PROGRAM PR_Line01
VAR PERSISTENT
//----------------VAR SETTING--------------------
	timerCheckCylinder_Up			: REAL;//CupSupply
	timerCheckCylinder_Dw			: REAL;
	timerCheckEmpty					: REAL;
	timerCheckStuck					: REAL;
	timerCylinder_Up_extend 		: REAL;
	timerCylinder_Suction_Cup_extend: REAL;
	timerCylinder_Suction_Cup		: REAL;
	timerCylinder_Suction_Val		: REAL;
	timerCylinder_Suction_pick		: REAL;
	fSpeed_motor_mixer				: REAL;//FoodMixer
	fTimer_Reverse					: REAL;
	fFast_Speed						: REAL;//FoodWeight
	fSlow_Speed_1					: REAL;
	fSlow_Speed_2					: REAL;
	fDerisedWeight_Food				: REAL;
	fChangeMode_Food_1				: REAL;
	fChangeMode_Food_2				: REAL;
	fMaxWeight_Food					: REAL;
	fPerStop_Food					: REAL;
	fTimer_Food						: REAL;
	fTimer_Alarm_Food				: REAL;
	fTimer_Check_Food				: REAL;
	fDelta_Food						: REAL;
	fTimer_rever_food				: REAL;
	fTimer_Error_Food				: REAL;
	fFast_Speed_vibrating_funnel	: REAL;//WormWeight
	fSlow_Speed_vibrating_funnel_1	: REAL;
	fSlow_Speed_vibrating_funnel_2	: REAL;
	fDerisedWeight_Worm				: REAL;
	fChangeMode_Worm_1				: REAL;
	fChangeMode_Worm_2				: REAL;
	fMaxWeight_Worm					: REAL;
	fPerStop_Worm					: REAL;
	fTimer_Worm						: REAL;
	fTimer_Alarm_Worm				: REAL;
	fTimer_Check_Worm				: REAL;
	fTimer_Check_Cylinder			: REAL;
	fDelta_Worm						: REAL;
	fTimer_Error_Worm				: REAL;
	timerCylinder_Suction			: REAL;//LidSupply
	timerCheckLidRelease			: REAL;
	timerLidBlow					: REAL;
	timerCheckLidEmpty				: REAL;
	timerCheckLidSuck				: REAL;
	timerCylinder_Stopper			: REAL;
	timer_Check_Cylinder_extend		: REAL;//LidClose
	timer_Check_Cylinder_retract	: REAL;
	timer_CloseLid					: REAL;
	fTimer_Comb						: REAL;//Transfer
	fTimer_Clip						: REAL;
	fTimer_Move_Comb				: REAL;
//-----------------VAR HMI-------------------
	fProductLog						: ARRAY [1..2] OF ARRAY  [1..5] OF REAL;
END_VAR

VAR
	bStatus_Food					: BOOL;
	bStatus_Worm					: BOOL;
//----------------VAR MANUAL---------------------
	bCylinder_up_extend 			: BOOL;//CupSupply
	bCylinder_up_retract 			: BOOL;
	bCylinder_dw_extend 			: BOOL;
	bCylinder_dw_retract 			: BOOL;
	bCylinder_Suction_cup_extend	: BOOL;
	bCylinder_Suction_cup_retract	: BOOL;
	bUp_Motor_Mixer					: BOOL;//FoodMixer
	bDown_Motor_Mixer				: BOOL;
	bMotor_mixer_Manual				: BOOL;
	bMotor_mixer_reverse			: BOOL;
	bUp_Food_Motor					: BOOL;//FoodWeight
	bDown_Food_Motor				: BOOL;
	bZero_Loadcell_Food				: BOOL;
	bMotor_Food						: BOOL;
	bMotor_Food_reverse				: BOOL;
	bUp_vibrating_funnel			: BOOL;//WormWeight
	bDown_vibrating_funnel			: BOOL;
	bZero_Loadcell_Worm				: BOOL;
	bCylinder_Block_Worm_Extend		: BOOL;
	bCylinder_Block_Worm_Retract	: BOOL;
	bMotor_vibrating_funnel			: BOOL;	
	bCylinder_LidStopper_extend 	: BOOL;//LidSupply
	bCylinder_LidStopper_retract 	: BOOL;
	bCylinder_Suction_extend		: BOOL;
	bCylinder_Suction_retract		: BOOL;
	bLidSuctionValve				: BOOL;
	bCupSuctionValve				: BOOL;
	bBlowValve						: BOOL;
	bCylinder_CloseLid_Extend		: BOOL;//LidClose
	bCylinder_CloseLid_Retract		: BOOL;
	bCylinder_Comb_Extend			: BOOL;//Transfer
	bCylinder_Comb_Retract			: BOOL;
	bCylinder_Clip_Extend			: BOOL;
	bCylinder_Clip_Retract			: BOOL;
	bCylinder_Move_Comb_Extend		: BOOL;
	bCylinder_Move_Comb_Retract		: BOOL;
//------------------fbmodule----------------
	fb_CupSupply	: FB_CupSupplyModule;
	fb_FoodMixer	: FB_FoodMixerModule;
	fb_FoodWeight	: FB_FoodWeightModule;
	fb_WormWeight	: FB_WormWeightModule;
	fb_LidSupply	: FB_LidSupplyModule;
	fb_LidClose		: FB_LidCloseModule;
	fb_Transfer		: FB_Transfer;
//---------------- VAR Method ---------------
	nState				: INT;
	nState_Dropcup		: INT;
	nState_Transfer		: INT;
	nState_FoodWeight	: INT;
	nState_WormWeight	: INT;
	nState_LidClose		: INT;
	nState_LidSupply	: INT;
	nDoneTransfer		: INT;
	nDoneTransferStop	: INT;
	tmp					: INT;
	bDoneTakeLid		: BOOL;
	bDoneTransfer		: BOOL;
	bDoneCupSupply		: BOOL;
	bDoneFoodWeight		: BOOL;
	bDoneWormWeight		: BOOL;
	bDoneLidSupply		: BOOL;
	bDoneLidClose		: BOOL;
	bEnable				: BOOL;
	bFinishCupSupply	: BOOL;
	bFinishFoodWeight	: BOOL;
	bFinishWormWeight	: BOOL;
	bFinishLidSupply	: BOOL;
	bFinishLidClose		: BOOL;
	bFinishTransfer		: BOOL;
	//-------VAR--------------
	nStateConveyor		: INT;
	fbtimertransfer		: TON;
	nStateStop			: INT;
	fbTimer				: ton;
	fbtimerStop			: ton;
	fbTimerCycle		: ton;
	timeCycle			: REAL :=1;
	fproduct			: INT;
	nstateCycle			: INT;
	bDone				: R_TRIG;
	fbDelay				: TON;
	bStatus_Food_order	: ARRAY [1..3] OF BOOL;
	bStatus_Worm_order	: ARRAY [1..3] OF BOOL;
	bStatus_Lid_order	: ARRAY [1..3] OF BOOL;
	i1,i2,i3			: INT := 0;
	xathucan			: BOOL;
	xasau				: BOOL;
	daothucan			: BOOL;
	transfer			: BOOL;
	nstatetest1			: INT;
	nstatetest2			: INT;
	nstatetest3			: INT;
	nstatetest4         : INT;
	bxa					: BOOL;
	bCheck				: BOOL;
	bypassfood			: BOOL;
	bypassWorm			: BOOL;
	bypassLid			: BOOL;
	eles: INT;
END_VAR

fb_CupSupply(
	nLine:= 1 , 
	timerCheckCylinder_Up:= timerCheckCylinder_Up, 
	timerCheckCylinder_Dw:= timerCheckCylinder_Dw, 
	timerCheckEmpty:= timerCheckEmpty, 
	timerCheckStuck:= timerCheckStuck,
	timerCylinder_Up_extend := timerCylinder_Up_extend,
	timerCylinder_Suction:= timerCylinder_Suction_Cup,
	timerCylinder_Suction_extend:= timerCylinder_Suction_Cup_extend,
	ttimerCylinder_val:= timerCylinder_Suction_Val,
	timerCylinder_Suction_pick:= timerCylinder_Suction_pick);

fb_FoodMixer(
	nLine:= 1,
	UnitID:= 4, 
	fSpeed_motor_mixer:= fSpeed_motor_mixer,
	fTimer_Reverse:= fTimer_Reverse);
		
fb_FoodWeight(
	nLine:= 1, 
	UnitID:= 7, 
	fFast_Speed:= fFast_Speed, 
	fSlow_Speed_1:= fSlow_Speed_1, 
	fSlow_Speed_2:= fSlow_Speed_2, 
	fDerisedWeight_Food:= fDerisedWeight_Food, 
	fChangeMode_Food_1:= fChangeMode_Food_1, 
	fChangeMode_Food_2:= fChangeMode_Food_2, 
	fMaxWeight_Food:= fMaxWeight_Food, 
	fPerStop_Food:= fPerStop_Food, 
	fTimer_Food:= fTimer_Food, 
	fTimer_Alarm_Food:= fTimer_Alarm_Food, 
	fTimer_Check_Food:= fTimer_Check_Food, 
	fDelta_Food:= fDelta_Food,
	fTimer_Reverse := fTimer_rever_food,
	fTimer_Error_Food := fTimer_Error_Food, 
	fProductLogF=> fProductLog[1],
	bStatus_Food=> bStatus_Food,
	Time_start => Time_Start_Food_line1,
	Time_Stop => Time_Stop_Food_line1,
	status=>bStatus_Food_line1,
	fweight_iot =>fWeight_food_line1);

fb_LidClose(
	nLine:= 1, 
	timer_Check_Cylinder_extend:= timer_Check_Cylinder_extend, 
	timer_Check_Cylinder_retract:= timer_Check_Cylinder_retract, 
	timer_CloseLid:= timer_CloseLid);
	
fb_LidSupply(
	nLine:= 1, 
	timerCylinder_Suction:= timerCylinder_Suction, 
	timerCheckLidRelease:= timerCheckLidRelease, 
	timerLidBlow:= timerLidBlow, 
	timerCheckLidEmpty:= timerCheckLidEmpty, 
	timerCheckLidSuck:= timerCheckLidSuck, 
	timerCylinder_Stopper:= timerCylinder_Stopper);

fb_Transfer(
	nLine:= 1, 
	fTimer_Comb:= fTimer_Comb, 
	fTimer_Clip:= fTimer_Clip, 
	fTimer_Move_Comb:= fTimer_Move_Comb, 
	nDoneTransfer=> nDoneTransfer,
	bDoneTransfer=> bDoneTransfer);

fb_WormWeight(
	nLine:= 1, 
	UnitID:= 5, 
	fFast_Speed_vibrating_funnel:= fFast_Speed_vibrating_funnel, 
	fSlow_Speed_vibrating_funnel_1:= fSlow_Speed_vibrating_funnel_1, 
	fSlow_Speed_vibrating_funnel_2:= fSlow_Speed_vibrating_funnel_2, 
	fDerisedWeight_Worm:= fDerisedWeight_Worm, 
	fChangeMode_Worm_1:= fChangeMode_Worm_1, 
	fChangeMode_Worm_2:= fChangeMode_Worm_2, 
	fMaxWeight_Worm:= fMaxWeight_Worm, 
	fPerStop_Worm:= fPerStop_Worm, 
	fTimer_Worm:= fTimer_Worm, 
	fTimer_Alarm_Worm:= fTimer_Alarm_Worm, 
	fTimer_Check_Worm:= fTimer_Check_Worm, 
	fTimer_Check_Cylinder:= fTimer_Check_Cylinder, 
	fDelta_Worm:= fDelta_Worm,
	fTimer_Error_Worm:= fTimer_Error_Worm, 
	fProductLog=> fProductLog[2],
	bStatus_Worm=>bStatus_Worm,
	Time_start=>Time_Start_Worm_line1,
	Time_Stop=>Time_Stop_Worm_line1,
	status=>bStatus_Worm_line1,
	fweight_iot =>fWeight_Worm_line1);

IF bClear1 THEN
	nResult_false1 := 0;
	nResult_true1 := 0;
	nCount1 := 0;
	bClear1 := FALSE;
END_IF	

fDerisedWeight_Food_line1	:= fDerisedWeight_Food;
fDerisedWeight_Worm_line1	:= fDerisedWeight_Worm;
fActDelta_Food_line1		:= fb_FoodWeight.fActDelta_Food;
fActDelta_Worm_line1		:= fb_WormWeight.fActDelta_Worm;
fDelta_Food_line1			:= fb_FoodWeight.fDelta_Food;
fDelta_Worm_line1			:= fb_WormWeight.fDelta_Worm;
	
IF getuser = 'Operator' THEN
	bypassfood := FALSE;
	bypassWorm := FALSE;
END_IF

ACTION Auto:
CASE nState OF
	0:// int
		bStatus_Food_order[1] := FALSE;
		bStatus_Worm_order[1] := FALSE;
		bStatus_Lid_order[1]  := FALSE;
		fb_Transfer.Init();
		fb_FoodWeight.SetZero();
		fb_WormWeight.SetZero();
		nDoneTransferStop	  := 0;
		i1 		:= 0;
		i2 		:= 0;
		i3 		:= 0;
		bfinish1	:= TRUE;
		nState 	:= 1;
		
	1: // Start
		nState_FoodWeight := 0;
		nState_WormWeight := 0;
		nState_LidSupply := 0;
		nState_LidClose := 0;
		bResetAuto1			:= FALSE;
		bDoneCupSupply 		:= FALSE;
		bDoneFoodWeight 	:= FALSE;
		bDoneWormWeight 	:= FALSE;
		bDoneLidSupply 		:= FALSE;
		bDoneLidClose 		:= FALSE;
		fb_FoodWeight.SetZero();
		fb_WormWeight.SetZero();
		nState := 11;
	11:
		bResetAuto1			:= FALSE;
		nState_Dropcup := 0;
		nState_Transfer := 0;
		bStop1 := FALSE;
		bShift_is_over1 := FALSE;
		bStatusStart1 := FALSE;
		fb_FoodMixer.Stop();
		nStatus1	:= 'STOP';
		bFinishCupSupply 	:= FALSE;
		bFinishFoodWeight 	:= FALSE;
		bFinishWormWeight	:= FALSE;
		bFinishLidSupply	:= FALSE;
		bFinishLidClose		:= FALSE;
		bFinishTransfer		:= FALSE;
		bfinish1	:= TRUE;
		nState := 22;
	22:
		IF bStart1 THEN
			bfinish1		:= FALSE;
			bStatusStart1 	:= TRUE;
			bToDropcup1 	:= FALSE;
			bResetAuto1		:= TRUE;
			status			:= 'RUN';
			nState := 2;
		END_IF
		
	2: // start mode auto
		bfinish1		:= FALSE;
		nStatus1	:= 'RUN';
		bResetAuto1		:= TRUE;
		bStart1 := FALSE;
		IF bypassfood THEN
			fb_FoodMixer.Stop();
		ELSE
			fb_FoodMixer.Auto();
		END_IF
		fb_CupSupply.CheckCup();
		fb_LidSupply.CheckLid();
		bDone(CLK := bDoneTransfer);
		CASE nstateCycle OF 
			0:
				fbTimerCycle(IN := TRUE, PT := T#100S);
				IF bDone.Q THEN
					nstateCycle := 1;
				END_IF
			1:
				timeCycle := TIME_TO_REAL(fbTimerCycle.ET)/1000;
				nstateCycle := 2;
			2: 
				fproduct :=  REAL_TO_INT(3600/(timeCycle+0.001));
				fbTimerCycle(IN := FALSE);
				nstateCycle := 0;
		END_CASE
		CASE nState_Dropcup OF
			0:// waiting for transfer
				fbDelay(IN := FALSE);
				fb_CupSupply.HoldCup();
				IF bToDropcup1 THEN
					nState_Dropcup := 1;
				END_IF
			1:// dropcup
				IF fb_CupSupply.DropCup() THEN
					bDoneCupSupply := TRUE;
					bToDropcup1 := FALSE;
					nState_Dropcup := 2;
				END_IF
			2:
				fbDelay(IN := TRUE, PT := T#300MS);
				IF fbDelay.Q THEN
					nState_Dropcup := 0;
				END_IF
		END_CASE
		
		CASE nState_FoodWeight OF
			0:// waiting for transfer
				IF bDoneTransfer THEN
					i1 := i1 + 1;
					fbTimer(IN := FALSE);
					nState_FoodWeight := 1;	
				END_IF
			1:// Check cup present
				IF NOT fb_FoodWeight.bIsCupPresent THEN
					IF bypassfood THEN
						nState_FoodWeight := 3;
						bStatus_Food_order[i1] := TRUE;
					ELSE
						nState_FoodWeight := 2;
					END_IF
				ELSE
					bStatus_Food_order[i1] := FALSE;
					nState_FoodWeight := 3;
				END_IF
			2:// FoodWeight
				IF NOT fb_FoodWeight.bIsCupPresent THEN
					IF fb_FoodWeight.Auto() THEN
						bStatus_Food_order[i1] := bStatus_Food;
						nState_FoodWeight := 3;
					END_IF
				ELSE
					nState_FoodWeight := 22;
				END_IF 
			22:
				fbTimer(IN := TRUE, PT := T#0.3S);
				fb_FoodWeight.Auto();
				IF fbTimer.Q THEN
					fb_FoodWeight.Init();
					nState_FoodWeight := 0;
				END_IF
			3:// check i
				IF i1 < 3 THEN
					nState_FoodWeight := 5;
				ELSE 
					i1 := 2;
					nState_FoodWeight := 4;
				END_IF
			4:// dao vi tri
				bStatus_Food_order[1] := bStatus_Food_order[2];
				bStatus_Food_order[2] := bStatus_Food_order[3];
				nState_FoodWeight := 5;
			5:// Done
				bDoneFoodWeight := TRUE;
				nState_FoodWeight := 10;
		END_CASE
		
		CASE nState_WormWeight OF
			0: // waiting for transfer
				IF bDoneTransfer THEN
					i2 := i2 + 1;;
					fbTimer(IN := FALSE);
					nState_WormWeight := 1;
				END_IF
			1:
				IF NOT fb_WormWeight.bIsCupPresent THEN
					nCount1 := nCount1 + 1;
					nState_WormWeight := 11;
				ELSE
					bStatus_Worm_order[i2] := FALSE;
					nState_WormWeight := 3;
				END_IF
			11: // check food
				IF bStatus_Food_order[1] THEN
					IF bypassWorm THEN
						nState_WormWeight := 3;
						bStatus_Worm_order[i2] := TRUE;
					ELSE
						nState_WormWeight := 2;
					END_IF
				ELSE
					bStatus_Worm_order[i2] := FALSE;
					nState_WormWeight := 3;
				END_IF	
			2:// WormWeight
				IF NOT fb_WormWeight.bIsCupPresent THEN
					IF fb_WormWeight.Auto() THEN
						bStatus_Worm_order[i2] := bStatus_Worm;
						nState_WormWeight := 3;
					END_IF
				ELSE
					nState_WormWeight := 22;
				END_IF
			22:
				fbTimer(IN := TRUE, PT := T#0.3S);
				fb_WormWeight.Auto(); 
				IF fbTimer.Q THEN
					fb_WormWeight.Init();
					nState_WormWeight := 0;
				END_IF
			3:// check i
				IF bStatus_Worm_order[i2] THEN
					nResult_true1 := nResult_true1 + 1;
				END_IF
				IF i2 < 3 THEN
					nState_WormWeight := 5;
				ELSE
					i2 := 2;
					nState_WormWeight := 4;
				END_IF
			4:// dao vi tri
				nResult_false1 := nCount1 - nResult_true1;
				bStatus_Worm_order[1] := bStatus_Worm_order[2];
				bStatus_Worm_order[2] := bStatus_Worm_order[3];
				nState_WormWeight 	  := 5;
			5:// Done 
				bDoneWormWeight       := TRUE;
				nState_WormWeight	  := 10;
		END_CASE
		
		CASE nState_LidSupply OF
			0:// waiting for transfer
				IF bDoneTransfer THEN
					i3 := i3 + 1;
					nState_LidSupply := 1;
				END_IF
			1:// check worm
				IF bStatus_Worm_order[1] THEN
					IF bypassLid THEN
						bStatus_Lid_order[i3] := FALSE;
						nState_LidSupply := 4;
					ELSE
						nState_LidSupply := 2;
					END_IF
				ELSE
					bStatus_Lid_order[i3] := FALSE;
					nState_LidSupply := 4;
				END_IF
			2:// take lid
				IF fb_LidSupply.TakeLid() THEN
					nState_LidSupply := 3;
				END_IF
			3:// drop lid
				IF fb_LidSupply.DropLid() THEN
					bStatus_Lid_order[i3] := TRUE;
					nState_LidSupply := 4;
				END_IF
			4:// check i
				IF i3 < 3 THEN
					nState_LidSupply := 6;
				ELSE
					i3 := 2;
					nState_LidSupply := 5;
				END_IF
			5:// dao vi tri
				bStatus_Lid_order[1] := bStatus_Lid_order[2];
				bStatus_Lid_order[2] := bStatus_Lid_order[3];
				nState_LidSupply 	 := 6;
			6:// Done
				bDoneLidSupply 		 := TRUE;
				nState_LidSupply 	 := 10;
		END_CASE
		
		CASE nState_LidClose OF
			0: // waiting for transfer
				IF bDoneTransfer THEN
					nState_LidClose := 1;
				END_IF
			1:// Check lid supply
				IF  bStatus_Lid_order[1] THEN
					nState_LidClose := 2;
				ELSE
					nState_LidClose := 3;
				END_IF
			2:// Close lid
				IF fb_LidClose.CloseLid() THEN
					nState_LidClose := 3;
				END_IF
			3://Done
				bDoneLidClose := TRUE;
				nState_LidClose := 10;
		END_CASE
		
		CASE nState_Transfer OF
			0:// waiting for Done module
				IF nDoneTransfer = 0 THEN
					nState_Transfer := 1;
				ELSIF nDoneTransfer > 0 THEN
					IF bDoneCupSupply AND bDoneFoodWeight AND bDoneWormWeight AND bDoneLidSupply AND bDoneLidClose THEN
						nState_Transfer := 1;
					END_IF
				END_IF
			1:
				IF fb_CupSupply.isCupDrop THEN
					bDoneCupSupply 	:= FALSE;
					bDoneFoodWeight := FALSE;
					bDoneWormWeight := FALSE;
					bDoneLidSupply 	:= FALSE;
					bDoneLidClose 	:= FALSE;
					nState_Transfer := 11;
				ELSE 
					F_SetError(2,nLine:=1);
				END_IF
			11:// transfer
				IF fb_Transfer.Auto() THEN
					nShoot1 := nShoot1 + 1; 
					nState_Transfer:= 2;
				END_IF
			2:
				nState_FoodWeight := 0;
				nState_WormWeight := 0;
				nState_LidSupply  := 0;
				nState_LidClose	  := 0;
				nState_Transfer	  := 0;
		END_CASE
		//Stop button
		IF bStop1 THEN
			nState := 3;
			bStartLine1 := FALSE;
		ELSIF bShift_is_over1 THEN
			nState := 4;
		END_IF
	3://Stop
		bfinish1 := FALSE;
		fb_CupSupply.CheckCup();
		fb_LidSupply.CheckLid();
		bResetAuto1		:= TRUE;
		nStatus1	:= 'RUN';
		IF bypassfood THEN
			fb_FoodMixer.Stop();
		ELSE
			fb_FoodMixer.Auto();
		END_IF
		CASE nState_Dropcup OF
			0:// waiting for transfer
				fbDelay(IN := FALSE);
				fb_CupSupply.HoldCup();
				IF bToDropcup1 THEN
					nState_Dropcup := 1;
				END_IF
				IF bFinishTransfer THEN
					nState_Dropcup := 10;
				END_IF
			1:// dropcup
				IF fb_CupSupply.DropCup() THEN
					bDoneCupSupply := TRUE;
					bToDropcup1 := FALSE;
					nState_Dropcup := 2;
				END_IF
			2:
				fbDelay(IN := TRUE, PT := T#300MS);
				IF fbDelay.Q THEN
					nState_Dropcup := 10;
				END_IF
			10:// finish
				bDoneCupSupply := TRUE;
				bFinishCupSupply := TRUE;
		END_CASE
		
		CASE nState_FoodWeight OF
			0:// waiting for transfer
				IF bDoneTransfer THEN
					i1 := i1 + 1;
					fbTimer(IN := FALSE);
					nState_FoodWeight := 1;	
				END_IF
			1:// Check cup present
				IF NOT fb_FoodWeight.bIsCupPresent THEN
					IF bypassfood THEN
						nState_FoodWeight := 3;
						bStatus_Food_order[i1] := TRUE;
					ELSE
						nState_FoodWeight := 2;
					END_IF
				ELSE
					bStatus_Food_order[i1] := FALSE;
					nState_FoodWeight := 3;
				END_IF
			2:// FoodWeight
				IF NOT fb_FoodWeight.bIsCupPresent THEN
					IF fb_FoodWeight.Auto() THEN
						bStatus_Food_order[i1] := bStatus_Food;
						nState_FoodWeight := 3;
					END_IF
				ELSE
					nState_FoodWeight := 22;
				END_IF 
			22:
				fbTimer(IN := TRUE, PT := T#0.3S);
				fb_FoodWeight.Auto();
				IF fbTimer.Q THEN
					fb_FoodWeight.Init();
					nState_FoodWeight := 0;
				END_IF
			3:// check i
				IF i1 < 3 THEN
					nState_FoodWeight := 5;
				ELSE 
					i1 := 2;
					nState_FoodWeight := 4;
				END_IF
			4:// dao vi tri
				bStatus_Food_order[1] := bStatus_Food_order[2];
				bStatus_Food_order[2] := bStatus_Food_order[3];
				nState_FoodWeight := 5;
			5:// Done
				bDoneFoodWeight := TRUE;
				nState_FoodWeight := 10;
			10:// finish
				bFinishFoodWeight := TRUE;
		END_CASE
		
		CASE nState_WormWeight OF
			0: // waiting for transfer
				IF bDoneTransfer THEN
					i2 := i2 + 1;;
					fbTimer(IN := FALSE);
					nState_WormWeight := 1;
				END_IF
			1:
				IF NOT fb_WormWeight.bIsCupPresent THEN
					nCount1 := nCount1 + 1;
					nState_WormWeight := 11;
				ELSE
					bStatus_Worm_order[i2] := FALSE;
					nState_WormWeight := 3;
				END_IF
			11: // check food
				IF bStatus_Food_order[1] THEN
					IF bypassWorm THEN
						nState_WormWeight := 3;
						bStatus_Worm_order[i2] := TRUE;
					ELSE
						nState_WormWeight := 2;
					END_IF
				ELSE
					bStatus_Worm_order[i2] := FALSE;
					nState_WormWeight := 3;
				END_IF	
			2:// WormWeight
				IF NOT fb_WormWeight.bIsCupPresent THEN
					IF fb_WormWeight.Auto() THEN
						bStatus_Worm_order[i2] := bStatus_Worm;
						nState_WormWeight := 3;
					END_IF
				ELSE
					nState_WormWeight := 22;
				END_IF
			22:
				fbTimer(IN := TRUE, PT := T#0.3S);
				fb_WormWeight.Auto(); 
				IF fbTimer.Q THEN
					fb_WormWeight.Init();
					nState_WormWeight := 0;
				END_IF
			3:// check i
				IF bStatus_Worm_order[i2] THEN
					nResult_true1 := nResult_true1 + 1;
				END_IF
				IF i2 < 3 THEN
					nState_WormWeight := 5;
				ELSE
					i2 := 2;
					nState_WormWeight := 4;
				END_IF
			4:// dao vi tri
				nResult_false1 := nCount1 - nResult_true1;
				bStatus_Worm_order[1] := bStatus_Worm_order[2];
				bStatus_Worm_order[2] := bStatus_Worm_order[3];
				nState_WormWeight 	  := 5;
			5:// Done 
				bDoneWormWeight       := TRUE;
				nState_WormWeight	  := 10;
			10:// finish
				bFinishWormWeight	  := TRUE;
		END_CASE
		
		CASE nState_LidSupply OF
			0:// waiting for transfer
				IF bDoneTransfer THEN
					i3 := i3 + 1;
					nState_LidSupply := 1;
				END_IF
			1:// check worm
				IF bStatus_Worm_order[1] THEN
					IF bypassLid THEN
						bStatus_Lid_order[i3] := FALSE;
						nState_LidSupply := 4;
					ELSE
						nState_LidSupply := 2;
					END_IF
				ELSE
					bStatus_Lid_order[i3] := FALSE;
					nState_LidSupply := 4;
				END_IF
			2:// take lid
				IF fb_LidSupply.TakeLid() THEN
					nState_LidSupply := 3;
				END_IF
			3:// drop lid
				IF fb_LidSupply.DropLid() THEN
					bStatus_Lid_order[i3] := TRUE;
					nState_LidSupply := 4;
				END_IF
			4:// check i
				IF i3 < 3 THEN
					nState_LidSupply := 6;
				ELSE
					i3 := 2;
					nState_LidSupply := 5;
				END_IF
			5:// dao vi tri
				bStatus_Lid_order[1] := bStatus_Lid_order[2];
				bStatus_Lid_order[2] := bStatus_Lid_order[3];
				nState_LidSupply 	 := 6;
			6:// Done
				bDoneLidSupply 		 := TRUE;
				nState_LidSupply 	 := 10;
			10:// finish
				bFinishLidSupply	 := TRUE;
		END_CASE
		
		CASE nState_LidClose OF
			0: // waiting for transfer
				IF bDoneTransfer THEN
					nState_LidClose := 1;
				END_IF
			1:// Check lid supply
				IF  bStatus_Lid_order[1] THEN
					nState_LidClose := 2;
				ELSE
					nState_LidClose := 3;
				END_IF
			2:// Close lid
				IF fb_LidClose.CloseLid() THEN
					nState_LidClose := 3;
				END_IF
			3://Done
				bDoneLidClose   := TRUE;
				nState_LidClose := 10;
			10:// finish
				bFinishLidClose := TRUE;
		END_CASE
		
		CASE nState_Transfer OF
			0:// waiting for Done module
				IF nDoneTransfer = 0 THEN
					nState_Transfer := 10;
				ELSIF nDoneTransfer > 0 THEN
					IF bDoneCupSupply AND bDoneFoodWeight AND bDoneWormWeight AND bDoneLidSupply AND bDoneLidClose THEN
					nState_Transfer := 10;
					END_IF
				END_IF
			1:
				IF fb_CupSupply.isCupDrop THEN
					bDoneCupSupply 	:= FALSE;
					bDoneFoodWeight := FALSE;
					bDoneWormWeight := FALSE;
					bDoneLidSupply 	:= FALSE;
					bDoneLidClose 	:= FALSE;
					nState_Transfer := 11;
				ELSE 
					F_SetError(2,nLine:=1);
				END_IF
			11:// transfer
				IF fb_Transfer.Auto() THEN
					nShoot1 := nShoot1 + 1;
					nState_Transfer:= 2;
				END_IF
			2: 
				nState_FoodWeight := 0;
				nState_WormWeight := 0;
				nState_LidSupply  := 0;
				nState_LidClose	  := 0;
				nState_Dropcup 	  := 0;
				nState_Transfer   := 0;
			10:// finish
				bFinishTransfer		:= TRUE;	
		END_CASE
		
		IF bFinishCupSupply AND bFinishFoodWeight AND bFinishWormWeight AND bFinishLidSupply AND bFinishLidClose AND bFinishTransfer THEN
			bfinish1	:= TRUE;
			nState := 11;
		END_IF
	4:// shift is over
		bfinish1 := FALSE;
		bStart1	:= FALSE;
		IF bypassfood THEN
			fb_FoodMixer.Stop();
		ELSE
			fb_FoodMixer.Auto();
		END_IF
		fb_CupSupply.CheckCup();
		fb_LidSupply.CheckLid();
		bResetAuto1		:= TRUE;
		bStatusStart1 := FALSE;
		nStatus1	:= 'RUN';
		bDone(CLK := bDoneTransfer);
		CASE nstateCycle OF 
			0:
				fbTimerCycle(IN := TRUE, PT := T#30S);
				IF bDone.Q THEN
					nstateCycle := 1;
				END_IF
			1:
				timeCycle := TIME_TO_REAL(fbTimerCycle.ET)/1000;
				nstateCycle := 2;
			2: 
				fproduct  := REAL_TO_INT(3600/(timeCycle+0.001));
				fbTimerCycle(IN := FALSE);
				nstateCycle := 0;
		END_CASE
		
		CASE nState_Dropcup OF
			0:// waiting for transfer
				fbDelay(IN := FALSE);
				fb_CupSupply.HoldCup();
				IF bToDropcup1 THEN
					nState_Dropcup := 10;
				END_IF
			1:// dropcup
				IF fb_CupSupply.DropCup() THEN
					bDoneCupSupply := TRUE;
					bToDropcup1 := FALSE;
					nState_Dropcup := 2;
				END_IF
			2:
				fbDelay(IN := TRUE, PT := T#300MS);
				IF fbDelay.Q THEN
					nState_Dropcup := 10;
				END_IF
			10:// finish
				bDoneCupSupply := TRUE;
				bFinishCupSupply := TRUE;
		END_CASE
		
		CASE nState_FoodWeight OF
			0:// waiting for transfer
				IF bDoneTransfer AND nDoneTransferStop < 4 THEN
					i1 := i1 + 1;
					fbTimer(IN := FALSE);
					nState_FoodWeight := 1;	
				ELSIF bDoneTransfer AND nDoneTransferStop >= 4 THEN
					i1 := i1 + 1;
					fbTimer(IN := FALSE);
					nState_FoodWeight := 33;	
				END_IF
			1:// Check cup present
				IF NOT fb_FoodWeight.bIsCupPresent THEN
					IF bypassfood THEN
						nState_FoodWeight := 3;
						bStatus_Food_order[i1] := TRUE;
					ELSE
						nState_FoodWeight := 2;
					END_IF
				ELSE
					bStatus_Food_order[i1] := FALSE;
					nState_FoodWeight := 3;
				END_IF
			2:// FoodWeight
				IF NOT fb_FoodWeight.bIsCupPresent THEN
					IF fb_FoodWeight.Auto() THEN
						bStatus_Food_order[i1] := bStatus_Food;
						nState_FoodWeight := 3;
					END_IF
				ELSE
					nState_FoodWeight := 22;
				END_IF 
			22:
				fbTimer(IN := TRUE, PT := T#0.3S);
				fb_FoodWeight.Auto();
				IF fbTimer.Q THEN
					fb_FoodWeight.Init();
					nState_FoodWeight := 0;
				END_IF
			33:
				bStatus_Food_order[i1] := FALSE;
				nState_FoodWeight := 3;
			3:// check i
				IF i1 < 3 THEN
					nState_FoodWeight := 5;
				ELSE 
					i1 := 2;
					nState_FoodWeight := 4;
				END_IF
			4:// dao vi tri
				bStatus_Food_order[1] := bStatus_Food_order[2];
				bStatus_Food_order[2] := bStatus_Food_order[3];
				nState_FoodWeight := 5;
			5:// Done
				bDoneFoodWeight := TRUE;
				nState_FoodWeight := 10;
			10:// finish
				bFinishFoodWeight := TRUE;
		END_CASE
		
		CASE nState_WormWeight OF
			0: // waiting for transfer
				IF bDoneTransfer AND nDoneTransferStop < 6 THEN
					i2 := i2 + 1;;
					fbTimer(IN := FALSE);
					nState_WormWeight := 1;
				ELSIF bDoneTransfer AND nDoneTransferStop >= 6 THEN
					i2 := i2 + 1;;
					fbTimer(IN := FALSE);
					nState_WormWeight := 33;
				END_IF
			1:
				IF NOT fb_WormWeight.bIsCupPresent THEN
					nCount1 := nCount1 + 1;
					nState_WormWeight := 11;
				ELSE
					bStatus_Worm_order[i2] := FALSE;
					nState_WormWeight := 3;
				END_IF
			11: // check food
				IF bStatus_Food_order[1] THEN
					IF bypassWorm THEN
						nState_WormWeight := 3;
						bStatus_Worm_order[i2] := TRUE;
					ELSE
						nState_WormWeight := 2;
					END_IF
				ELSE
					bStatus_Worm_order[i2] := FALSE;
					nState_WormWeight := 3;
				END_IF	
			2:// WormWeight
				IF NOT fb_WormWeight.bIsCupPresent THEN
					IF fb_WormWeight.Auto() THEN
						bStatus_Worm_order[i2] := bStatus_Worm;
						nState_WormWeight := 3;
					END_IF
				ELSE
					nState_WormWeight := 22;
				END_IF
			22:
				fbTimer(IN := TRUE, PT := T#0.3S);
				fb_WormWeight.Auto(); 
				IF fbTimer.Q THEN
					fb_WormWeight.Init();
					nState_WormWeight := 0;
				END_IF
			33:
				bStatus_Worm_order[i2] := FALSE;
				nState_WormWeight := 3;
			3:// check i
				IF bStatus_Worm_order[i2] THEN
					nResult_true1 := nResult_true1 + 1;
				END_IF
				IF i2 < 3 THEN
					nState_WormWeight := 5;
				ELSE
					i2 := 2;
					nState_WormWeight := 4;
				END_IF
			4:// dao vi tri
				nResult_false1 := nCount1 - nResult_true1;
				bStatus_Worm_order[1] := bStatus_Worm_order[2];
				bStatus_Worm_order[2] := bStatus_Worm_order[3];
				nState_WormWeight 	  := 5;
			5:// Done 
				bDoneWormWeight       := TRUE;
				nState_WormWeight	  := 10;
			10:// finish
				bFinishWormWeight	  := TRUE;
		END_CASE
		
		CASE nState_LidSupply OF
			0:// waiting for transfer
				IF bDoneTransfer THEN
					i3 := i3 + 1;
					nState_LidSupply := 1;
				END_IF
			1:// check worm
				IF bStatus_Worm_order[1] THEN
					IF bypassLid THEN
						bStatus_Lid_order[i3] := FALSE;
						nState_LidSupply := 4;
					ELSE
						nState_LidSupply := 2;
					END_IF
				ELSE
					bStatus_Lid_order[i3] := FALSE;
					nState_LidSupply := 4;
				END_IF
			2:// take lid
				IF fb_LidSupply.TakeLid() THEN
					nState_LidSupply := 3;
				END_IF
			3:// drop lid
				IF fb_LidSupply.DropLid() THEN
					bStatus_Lid_order[i3] := TRUE;
					nState_LidSupply := 4;
				END_IF
			4:// check i
				IF i3 < 3 THEN
					nState_LidSupply := 6;
				ELSE
					i3 := 2;
					nState_LidSupply := 5;
				END_IF
			5:// dao vi tri
				bStatus_Lid_order[1] := bStatus_Lid_order[2];
				bStatus_Lid_order[2] := bStatus_Lid_order[3];
				nState_LidSupply 	 := 6;
			6:// Done
				bDoneLidSupply 		 := TRUE;
				nState_LidSupply 	 := 10;
			10:// finish
				bFinishLidSupply	 := TRUE;
		END_CASE
		
		CASE nState_LidClose OF
			0: // waiting for transfer
				IF bDoneTransfer THEN
					nState_LidClose := 1;
				END_IF
			1:// Check lid supply
				IF  bStatus_Lid_order[1] THEN
					nState_LidClose := 2;
				ELSE
					nState_LidClose := 3;
				END_IF
			2:// Close lid
				IF fb_LidClose.CloseLid() THEN
					nState_LidClose := 3;
				END_IF
			3://Done
				bDoneLidClose   := TRUE;
				nState_LidClose := 10;
			10:// finish
				bFinishLidClose := TRUE;
		END_CASE
		
		CASE nState_Transfer OF
			0:// waiting for Done module
				IF bDoneCupSupply AND bDoneFoodWeight AND bDoneWormWeight AND bDoneLidSupply AND bDoneLidClose THEN
					nState_Transfer := 1;
				END_IF
			1:
				IF fb_CupSupply.isCupDrop THEN
					bDoneCupSupply 	:= FALSE;
					bDoneFoodWeight := FALSE;
					bDoneWormWeight := FALSE;
					bDoneLidSupply 	:= FALSE;
					bDoneLidClose 	:= FALSE;
					nState_Transfer := 11;
				ELSE 
					F_SetError(2,nLine:=1);
				END_IF
			11:// transfer
				IF fb_Transfer.Auto() THEN
					nShoot1 := nShoot1 + 1;
					nState_Transfer:= 2;
				END_IF
			2:
				nState_FoodWeight := 0;
				nState_WormWeight := 0;
				nState_LidSupply  := 0;
				nState_LidClose	  := 0;
				nDoneTransferStop := nDoneTransferStop + 1;
				nState_Transfer   := 3;
			3:
				IF nDoneTransferStop < 11 THEN
					nState_Transfer   := 0;
				ELSE
					nState_Transfer   := 10;
				END_IF
			10:// finish
				bFinishTransfer		:= TRUE;
		END_CASE
		IF bFinishCupSupply AND bFinishFoodWeight AND bFinishWormWeight AND bFinishLidSupply AND bFinishLidClose AND bFinishTransfer THEN
			bfinish1	:= TRUE;
			nState := 0;
		END_IF
END_CASE
END_ACTION

ACTION check:
IF fb_CupSupply.fbCylinder_Up.bIsRetract THEN
	bCylinder_up_retract 	:= TRUE;
	bCylinder_up_extend		:= FALSE;
ELSE
	bCylinder_up_retract 	:= FALSE;
	bCylinder_up_extend		:= TRUE;
END_IF

IF fb_CupSupply.fbCylinder_Dw.bIsExtend THEN
	bCylinder_dw_extend 	:= TRUE;
	bCylinder_dw_retract 	:= FALSE;
ELSIF fb_CupSupply.fbCylinder_Dw.bIsRetract THEN
	bCylinder_dw_extend 	:= FALSE;
	bCylinder_dw_retract 	:= TRUE;
ELSE
	bCylinder_dw_extend 	:= FALSE;
	bCylinder_dw_retract 	:= FALSE;
END_IF

IF fb_CupSupply.fbCylinder_Suction.bIsExtend THEN
	bCylinder_Suction_cup_extend 	:= TRUE;
	bCylinder_Suction_cup_retract	:= FALSE;
ELSE
	bCylinder_Suction_cup_extend 	:= FALSE;
	bCylinder_Suction_cup_retract	:= TRUE;
END_IF
//--------------------------------------
IF fb_WormWeight.fbCylinder.bIsRetract THEN
	bCylinder_Block_Worm_Extend	 := FALSE;
	bCylinder_Block_Worm_Retract := TRUE;
ELSE
	bCylinder_Block_Worm_Extend	 := TRUE;
	bCylinder_Block_Worm_Retract := FALSE;
END_IF
//--------------------------------------
IF fb_LidSupply.fbCylinder_LidStopper.bIsExtend THEN
	bCylinder_LidStopper_extend 	:= TRUE;
	bCylinder_LidStopper_retract 	:= FALSE;
ELSIF fb_LidSupply.fbCylinder_LidStopper.bIsRetract THEN
	bCylinder_LidStopper_extend 	:= FALSE;
	bCylinder_LidStopper_retract 	:= TRUE;
ELSE
	bCylinder_LidStopper_extend 	:= FALSE;
	bCylinder_LidStopper_retract 	:= FALSE;
END_IF

IF fb_LidSupply.fbCylinder_Suction.bIsExtend THEN
	bCylinder_Suction_extend		:= TRUE;
	bCylinder_Suction_retract		:= FALSE;
ELSIF fb_LidSupply.fbCylinder_Suction.bIsRetract THEN
	bCylinder_Suction_extend		:= FALSE;
	bCylinder_Suction_retract		:= TRUE;
ELSE
	bCylinder_Suction_extend		:= FALSE;
	bCylinder_Suction_retract		:= FALSE;
END_IF
//--------------------------------------
IF fb_LidClose.fbCylinder_LidClose.bIsExtend THEN
	bCylinder_CloseLid_Extend		:= TRUE;
	bCylinder_CloseLid_Retract		:= FALSE;
ELSIF fb_LidClose.fbCylinder_LidClose.bIsRetract THEN
	bCylinder_CloseLid_Extend		:= FALSE;
	bCylinder_CloseLid_Retract		:= TRUE;
ELSE
	bCylinder_CloseLid_Extend		:= FALSE;
	bCylinder_CloseLid_Retract		:= FALSE;
END_IF
//--------------------------------------
IF fb_Transfer.fbCylinder_Comb.bIsExtend THEN
	bCylinder_Comb_Extend			:= TRUE;
	bCylinder_Comb_Retract			:= FALSE;
ELSIF fb_Transfer.fbCylinder_Comb.bIsRetract THEN
	bCylinder_Comb_Extend			:= FALSE;
	bCylinder_Comb_Retract			:= TRUE;
ELSE
	bCylinder_Comb_Extend			:= FALSE;
	bCylinder_Comb_Retract			:= FALSE;
END_IF

IF fb_Transfer.fbCylinder_Clip.bIsExtend THEN
	bCylinder_Clip_Extend			:= TRUE;
	bCylinder_Clip_Retract			:= FALSE;
ELSIF fb_Transfer.fbCylinder_Clip.bIsRetract THEN
	bCylinder_Clip_Extend			:= FALSE;
	bCylinder_Clip_Retract			:= TRUE;
ELSE
	bCylinder_Clip_Extend			:= FALSE;
	bCylinder_Clip_Retract			:= FALSE;
END_IF

IF fb_Transfer.fbCylinder_Move_Comb.bIsExtend THEN
	bCylinder_Move_Comb_Extend		:= TRUE;
	bCylinder_Move_Comb_Retract		:= FALSE;
ELSIF fb_Transfer.fbCylinder_Move_Comb.bIsRetract THEN
	bCylinder_Move_Comb_Extend		:= FALSE;
	bCylinder_Move_Comb_Retract		:= TRUE;
ELSE
	bCylinder_Move_Comb_Extend		:= FALSE;
	bCylinder_Move_Comb_Retract		:= FALSE;
END_IF

bMotor_mixer_Manual				:= FALSE;
bMotor_mixer_reverse			:= FALSE;
bMotor_Food						:= FALSE;
bMotor_Food_reverse				:= FALSE;
bMotor_vibrating_funnel			:= FALSE;
END_ACTION

ACTION Check_reset:
IF fb_CupSupply.fbCylinder_Up.bIsRetract AND fb_CupSupply.fbCylinder_Dw.bIsExtend 
	AND NOT fb_WormWeight.fbCylinder.bIsRetract AND fb_LidSupply.fbCylinder_Suction.bIsRetract 
	AND fb_LidClose.fbCylinder_LidClose.bIsRetract AND fb_Transfer.fbCylinder_Comb.bIsRetract 
	AND fb_Transfer.fbCylinder_Clip.bIsRetract AND fb_Transfer.fbCylinder_Move_Comb.bIsRetract
	AND fb_CupSupply.fbCylinder_Suction.bIsExtend THEN
		bResetmanual1 := TRUE;
ELSE 
		bResetmanual1 := FALSE;
END_IF
IF bReset THEN
	bCylinder_up_retract 	:= TRUE;
	bCylinder_up_extend		:= FALSE;
	bCylinder_dw_extend 	:= TRUE;
	bCylinder_dw_retract 	:= FALSE;
	bCylinder_Suction_cup_retract 	:= FALSE;
	bCylinder_Suction_cup_extend 	:= TRUE;
	bCylinder_Block_Worm_Extend	 := TRUE;
	bCylinder_Block_Worm_Retract := FALSE;
	bCylinder_Suction_extend		:= FALSE;
	bCylinder_Suction_retract		:= TRUE;
	bCylinder_CloseLid_Extend		:= FALSE;
	bCylinder_CloseLid_Retract		:= TRUE;
	bCylinder_Comb_Extend			:= FALSE;
	bCylinder_Comb_Retract			:= TRUE;
	bCylinder_Clip_Extend			:= FALSE;
	bCylinder_Clip_Retract			:= TRUE;
	IF fb_Transfer.fbCylinder_Comb.bIsRetract THEN
		bCylinder_Move_Comb_Extend		:= FALSE;
		bCylinder_Move_Comb_Retract		:= TRUE;
	END_IF
	bxa := FALSE;
END_IF
END_ACTION

ACTION Init:
fb_CupSupply.Init();
fb_FoodWeight.Init();
fb_WormWeight.Init();
fb_LidSupply.Init();
fb_LidClose.Init();
fb_Transfer.Init();

nState := 0;
nState_Dropcup := 0;
nState_FoodWeight := 0;
nState_WormWeight := 0;
nState_LidSupply := 0;
nState_LidClose := 0;
nState_Transfer := 0;

bFinishCupSupply 	:= FALSE;
bFinishFoodWeight 	:= FALSE;
bFinishWormWeight	:= FALSE;
bFinishLidSupply	:= FALSE;
bFinishLidClose		:= FALSE;
bFinishTransfer		:= FALSE;

bDoneCupSupply 		:= FALSE;
bDoneFoodWeight 	:= FALSE;
bDoneWormWeight 	:= FALSE;
bDoneLidSupply 		:= FALSE;
bDoneLidClose 		:= FALSE;
bDoneTransfer		:= FALSE;
nDoneTransferStop	  := 0;

bStatus_Food_order[1] := FALSE;
bStatus_Worm_order[1] := FALSE;
bStatus_Lid_order[1]  := FALSE;
		
i1 		:= 0;
i2 		:= 0;
i3 		:= 0;
END_ACTION

ACTION Manual:
fb_CupSupply.Manual(bCylinder_dw_extend := bCylinder_dw_extend, bCylinder_dw_retract := bCylinder_dw_retract,
					bCylinder_up_extend := bCylinder_up_extend, bCylinder_up_retract := bCylinder_up_retract,
					bCylinder_suction_extend:= bCylinder_Suction_cup_extend, bCylinder_suction_retract := bCylinder_Suction_cup_retract);

IF bxa THEN
	IF daothucan THEN
		fb_FoodMixer.Auto();
	ELSE
		fb_FoodMixer.Stop();
	END_IF
ELSE
	daothucan := FALSE;	
	fb_FoodMixer.Manual(bDown_Motor_Mixer := bDown_Motor_Mixer, bUp_Motor_Mixer := bUp_Motor_Mixer,
					bMotor_mixer_Manual := bMotor_mixer_Manual,bMotor_mixer_reverse := bMotor_mixer_reverse);

	IF bUp_Motor_Mixer THEN
		bUp_Motor_Mixer := FALSE;
	END_IF
	
	IF bDown_Motor_Mixer THEN
		bDown_Motor_Mixer := FALSE;
	END_IF
END_IF

IF bxa THEN
	CASE nstatetest1 OF 
	0:
		IF xathucan THEN
			nstatetest1 := 1;			
		END_IF
	1:
		IF fb_FoodWeight.Auto() THEN
			nstatetest1 := 2;
		END_IF
	2: 
		xathucan := FALSE;
		nstatetest1 := 3;
	3:
		nstatetest1 := 0;
	END_CASE
ELSE
	xathucan := FALSE;
	nstatetest1 := 0;
	fb_FoodWeight.Manual(bDown_Food_Motor := bDown_Food_Motor, bUp_Food_Motor := bUp_Food_Motor,
									bMotor_Food := bMotor_Food, bZero_Loadcell_Food := bZero_Loadcell_Food, bMotor_Food_Reverse := bMotor_Food_reverse);
				
	IF bUp_Food_Motor THEN
		bUp_Food_Motor := FALSE;
	END_IF
				
	IF bDown_Food_Motor THEN
		bDown_Food_Motor := FALSE;
	END_IF
				
	IF bZero_Loadcell_Food THEN
		bZero_Loadcell_Food := FALSE;
	END_IF
END_IF

IF bxa THEN
	CASE nstatetest2 OF 
	0:
		IF xasau THEN
			nstatetest2 := 1;
		END_IF
	1:
		IF fb_WormWeight.Auto() THEN
			nstatetest2 := 2;
		END_IF
	2: 
		xasau := FALSE;
		nstatetest2 := 3;
	3:
		nstatetest2 := 0;
	END_CASE
ELSE
	xasau := FALSE;
	nstatetest2 := 0;
	fb_WormWeight.Manual(bCylinder_Block_Worm_Extend := bCylinder_Block_Worm_Extend, bCylinder_Block_Worm_Retract := bCylinder_Block_Worm_Retract,
					bDown_vibrating_funnel := bDown_vibrating_funnel, bUp_vibrating_funnel := bUp_vibrating_funnel,
					bMotor_vibrating_funnel := bMotor_vibrating_funnel, bZero_Loadcell_Worm := bZero_Loadcell_Worm);
	
	IF bUp_vibrating_funnel THEN
		bUp_vibrating_funnel := FALSE;
	END_IF
	
	IF bDown_vibrating_funnel THEN
		bDown_vibrating_funnel := FALSE;
	END_IF
	
	IF bZero_Loadcell_Worm THEN
		bZero_Loadcell_Worm := FALSE;
	END_IF
END_IF

fb_LidSupply.Manual(bCylinder_LidStopper_extend := bCylinder_LidStopper_extend, bCylinder_LidStopper_retract := bCylinder_LidStopper_retract,
					bCylinder_Suction_extend := bCylinder_Suction_extend, bCylinder_Suction_retract := bCylinder_Suction_retract,
					bCupSuctionValve := bCupSuctionValve, bLidSuctionValve := bLidSuctionValve, bBlowValve := bBlowValve);

fb_LidClose.Manual(bCylinder_CloseLid_Extend := bCylinder_CloseLid_Extend, bCylinder_CloseLid_Retract := bCylinder_CloseLid_Retract);



fb_Transfer.Manual(bCylinder_Clip_Extend := bCylinder_Clip_Extend, bCylinder_Clip_Retract := bCylinder_Clip_Retract,
				   bCylinder_Comb_Extend := bCylinder_Comb_Extend, bCylinder_Comb_Retract := bCylinder_Comb_Retract,
				   bCylinder_Move_Comb_Extend := bCylinder_Move_Comb_Extend, bCylinder_Move_Comb_Retract := bCylinder_Move_Comb_Retract);

IF fb_CupSupply.fbCylinder_Suction.bIsExtend AND fb_LidSupply.fbCylinder_Suction.bIsRetract AND fb_LidClose.fbCylinder_LidClose.bIsRetract THEN
	bCheck := TRUE;
ELSE
	bCheck := FALSE;
END_IF
END_ACTION

ACTION Reset:
fb_CupSupply.Reset();
fb_FoodMixer.Reset();
fb_FoodWeight.Reset();
fb_WormWeight.Reset();
fb_LidSupply.Reset();
fb_LidClose.Reset();
fb_Transfer.Reset();
nState := 22;
END_ACTION

ACTION Stop:
fb_FoodWeight.Stop();
fb_WormWeight.Stop();
fb_LidSupply.Stop();
fb_LidClose.Stop();
fb_Transfer.Stop();
fb_CupSupply.Stop();
bLidSuctionValve		:= FALSE;
bCupSuctionValve		:= FALSE;
bResetAuto1				:= FALSE;
fb_FoodMixer.Stop();
END_ACTION

END_PROGRAM

(* stored: Version 1.1.0.1, ProductVersion 3.1.4024.12
   POU PR_Line01: Id {d0ff51a4-eb4c-4ee0-a023-040919afc1d2}, SpecialFunc None
   Action Auto: Id {d2f01b4d-b3e1-4231-8308-415c05872c14}
   Action check: Id {eec90b22-ac29-461f-b299-7b3cfc6f0486}
   Action Check_reset: Id {365f44e1-62d3-4cb1-bea5-9baa2bb61b6b}
   Action Init: Id {c31d6c2c-6a8e-4683-acdd-a2d63b564f3e}
   Action Manual: Id {3cf3e0d2-17bd-450b-b8f2-6214979a1615}
   Action Reset: Id {28858929-868d-41c4-9c4e-1446ea304b31}
   Action Stop: Id {4ffacfa3-f561-4841-a5f4-feede6e91599} *)
